FUNCTION_BLOCK Heater
VAR_INPUT
	iWaterTemp : REAL;
END_VAR
VAR_OUTPUT
	oHeaterEnable : BOOL;
	oHeaterPower : REAL;
END_VAR
VAR_IN_OUT
	ioHeatStruct : THeater;
END_VAR
VAR
	pidParameters : ST_CTRL_PID_PARAMS;
END_VAR

pidParameters.fKp := 10; //P
pidParameters.tTn := T#2S; //I
pidParameters.tTv := T#0.5S; //D
pidParameters.tCtrlCycleTime := T#200MS;
pidParameters.tTaskCycleTime := T#100MS;
pidParameters.fOutMaxLimit := 100;
pidParameters.fOutMinLimit := 0;
pidParameters.bDInTheFeedbackPath := FALSE;
pidParameters.bPInTheFeedbackPath := FALSE;
pidParameters.bARWOnIPartOnly := FALSE;
pidParameters.tTd := T#100MS; 

ioHeatStruct.PID(
	fSetpointValue := ioHeatStruct.ParamHeatingSetPointAutomat, 
	fActualValue := iWaterTemp, 
	fManSyncValue := ioHeatStruct.ParamHeatingPowerManual,
	bSync := ioHeatStruct.State.ManCtrl,
	eMode := E_CTRL_MODE.eCTRL_MODE_ACTIVE, // automatic mode of PID component
	stParams := pidParameters);

ioHeatStruct.State.HeatingOut := ioHeatStruct.PID.fOut;

	 
{region "Manual/Automat"}
// switching state of engine - automatic or manual control (default state is manual)
	IF ioHeatStruct.Cmd.ManCtrl OR ioHeatStruct.State.GenErr THEN 
		ioHeatStruct.State.ManCtrl := TRUE;	  
		ioHeatStruct.State.AutCtrl := FALSE;
	END_IF
		 
	IF ioHeatStruct.Cmd.AutCtrl  AND NOT ioHeatStruct.Cmd.ManCtrl AND NOT ioHeatStruct.State.GenErr THEN
		ioHeatStruct.State.AutCtrl := TRUE;	 
		ioHeatStruct.State.ManCtrl := FALSE; 
	END_IF
		 
	IF  ioHeatStruct.State.AutCtrl  = ioHeatStruct.State.ManCtrl THEN 
		ioHeatStruct.State.AutCtrl := FALSE;	 
		ioHeatStruct.State.ManCtrl := TRUE; 
	END_IF
		 
	ioHeatStruct.Cmd.ManCtrl := FALSE;
	ioHeatStruct.Cmd.AutCtrl := FALSE;

{endregion}
	 
 
{region "ManCtrl"}
// processing manual actions - if command is processed, it is set to FALSE even if can't be processed
// Engine commands are turn off (stop) and turn on (start)
IF ioHeatStruct.State.ManCtrl  	THEN
	
	IF ioHeatStruct.Cmd.TurnOnMan	THEN
		ioHeatStruct.State.EnableOut	:= TRUE;
		END_IF	
	IF	ioHeatStruct.Cmd.TurnOffMan	THEN
		ioHeatStruct.State.EnableOut	:= FALSE;
		END_IF	
	IF	ioHeatStruct.Cmd.TurnOffMan =  ioHeatStruct.Cmd.TurnOnMan	THEN
		ioHeatStruct.State.EnableOut	:= FALSE;
		END_IF	
						   
END_IF
		

{endregion}
 
{region "AutCtrl"}
//if request to run in automatic mode set outputs to right states if MAR
//AutoRequest shouldn't be reseted to false state

{endregion}
 
{region "Error states"}
ioHeatStruct.ParamHeatingSetPointAutomat	:= 90;
{endregion}
// if water temperature is too high, stop heating and generate error
	IF iWaterTemp > ioHeatStruct.ParamHeatingSetPointAutomat THEN
		ioHeatStruct.State.Err := TRUE;
		oHeaterEnable := FALSE;
	END_IF
	 
{endregion}
	 
 
oHeaterPower := ioHeatStruct.State.HeatingOut;
oHeaterEnable := ioHeatStruct.State.EnableOut;

END_FUNCTION_BLOCK

(* stored: Version 1.1.0.1, ProductVersion 3.1.4024.15
   POU Heater: Id {fe81cd62-8fb3-4eb5-8579-8abf8e5327d3}, SpecialFunc None *)
